ABB RobotStudio station: Vision_HG_20250724-224039.rsstn

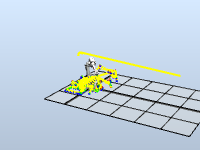
Station Station (saved by RobotStudio 6.8.8148.134)
Controller Vision
  mechanical unit ROB_1: IRB2600_20_165_C_01_2, 6 joints, base frame (0, 0, 0) mm
Layout (positions relative to the parent item):
  - IRB2600_20_165_C_01_2 [mechanism, from Robots\IRB2600_20_165_C_01.rslib] at (0, 0, 0) mm; joint values [-0.7369, -0.204, 0.6129, 0.0001, 1.0987, -0.0243] (rad or m)
  - 框架_2 [frame] at (695.76, -308.93, 242.8) mm, rotated rx -4.43 ry -84.98 rz 46.15 deg
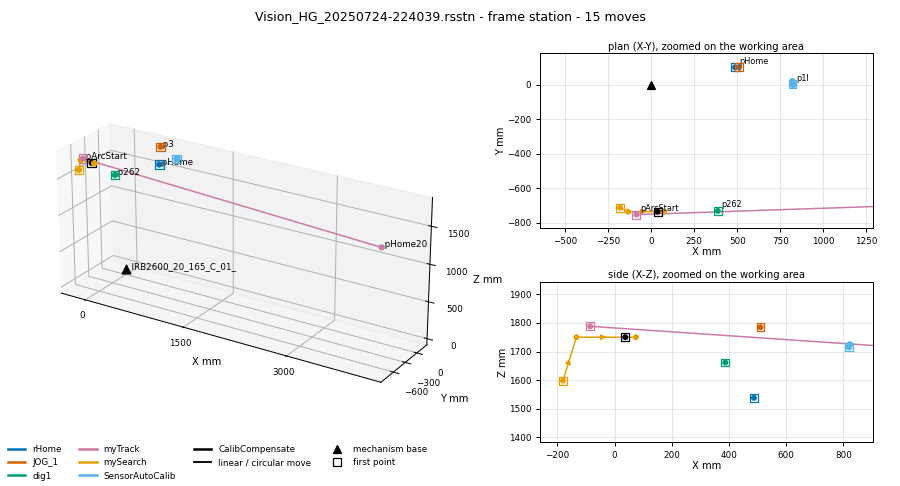
[picture p0: tool path of Vision_HG_20250724-224039.rsstn in frame station, 15 of 295 moves have a stored position in this frame; points joined in program order, loops and branches not executed]
Targets, tools, work objects and paths stored in the station, written as RAPID:
! task T_ROB1
MODULE MainModule
  VAR tooldata p1:=[TRUE,[[0,0,0],[1,0,0,0]],[-1,[0,0,0],[1,0,0,0],0,0,0]];
  LOCAL PERS tooldata p0:=[TRUE,[[0,0,0],[1,0,0,0]],[-1,[0,0,0],[1,0,0,0],0,0,0]];
  PERS tooldata tool3:=[TRUE,[[-77.6624,-1.03018,498.161],[0.800252,-0.0129489,0.0443032,-0.597884]],[10,[79.1,25.2,-267.1],[1,0,0,0],0.143,0.365,0.104]];
  TASK PERS tooldata tool4:=[TRUE,[[0,0,0],[1,0,0,0]],[10,[0,0,0],[1,0,0,0],0,0,0]];
  PERS tooldata tWeldGun:=[TRUE,[[-80.9134,-12.7311,494.27],[0.800252,-0.0129489,0.0443032,-0.597884]],[10,[79.1,25.2,-267.1],[1,0,0,0],0.143,0.365,0.104]];
  PERS tooldata autoCalibRes:=[TRUE,[[-92.3529,67.6081,476.661],[0.14635,-0.09099,-0.47804,-0.86127]],[2,[1,0,0],[1,0,0,0],0,0,0]];
  TASK PERS tooldata tool1:=[TRUE,[[0,0,0],[1,0,0,0]],[-1,[0,0,0],[1,0,0,0],0,0,0]];
  PERS wobjdata wobjcalib:=[FALSE,TRUE,"",[[826.111,71.2533,1714.68],[0.0119558,0.680715,0.732448,-0.00181828]],[[0,0,0],[1,0,0,0]]];
  CONST robtarget pHome:=[[487.33,102.53,1537.96],[0.139151,0.929573,0.0802124,-0.331809],[0,-1,0,1],[165.238,9E+09,9E+09,9E+09,9E+09,9E+09]];
  CONST speeddata speed1:=[25,25,25,25];
  CONST robtarget p3:=[[510.37,102.54,1784.95],[0.139155,0.929576,0.0802308,-0.331793],[0,-1,0,1],[165.238,9E+09,9E+09,9E+09,9E+09,9E+09]];
  CONST robtarget p262:=[[387.21,-731.34,1661.4],[0.0489836,0.0684608,0.2747,-0.957838],[0,0,-1,1],[276.422,9E+09,9E+09,9E+09,9E+09,9E+09]];
  PERS robtarget pArcStart:=[[-85.4083,-752.512,1788.13],[0.0516116,0.0583127,0.355092,-0.931582],[-1,-1,0,1],[443.838,9E+09,9E+09,9E+09,9E+09,9E+09]];
  CONST robtarget pHome20:=[[4100.11,-610.56,1504.11],[0.0519254,0.0584219,0.355084,-0.931561],[-1,-1,-1,1],[4151.67,9E+09,9E+09,9E+09,9E+09,9E+09]];
  CONST robtarget pBegin:=[[-180.6,-712.13,1598.38],[0.0515906,0.0582196,0.355192,-0.931551],[-1,-1,0,1],[443.838,9E+09,9E+09,9E+09,9E+09,9E+09]];
  PERS robtarget pSearchStart:=[[-133.62,-735.71,1750.06],[0.0516116,0.0583127,0.355092,-0.931582],[-1,-1,0,1],[443.838,9E+09,9E+09,9E+09,9E+09,9E+09]];
  PERS robtarget pSearchEnd:=[[74.4,-735.66,1750.11],[0.0517009,0.0583963,0.355037,-0.931593],[-1,-1,0,1],[443.838,9E+09,9E+09,9E+09,9E+09,9E+09]];
  CONST robtarget p1l:=[[-66.95,-10.33,0.38],[0.0609234,-0.0589398,-0.990074,0.112108],[-2,-1,2,1],[1474.6,9E+09,9E+09,9E+09,9E+09,9E+09]];
  CONST robtarget p2l:=[[-56.82,-10.34,0.37],[0.0609473,-0.0589005,-0.990073,0.112123],[-2,-1,2,1],[1474.6,9E+09,9E+09,9E+09,9E+09,9E+09]];
  CONST robtarget p3l:=[[-46.82,-10.3,0.33],[0.0609635,-0.0588963,-0.990075,0.112097],[-2,-1,2,1],[1474.6,9E+09,9E+09,9E+09,9E+09,9E+09]];
  CONST robtarget p1h:=[[-74.01,-7.93,-8.85],[0.0610072,-0.0589652,-0.990068,0.112102],[-2,-1,2,1],[1474.6,9E+09,9E+09,9E+09,9E+09,9E+09]];
  CONST robtarget p2h:=[[-63.94,-7.93,-8.86],[0.0610143,-0.0589296,-0.99007,0.112101],[-2,-1,2,1],[1474.6,9E+09,9E+09,9E+09,9E+09,9E+09]];
  CONST robtarget p3h:=[[-53.65,-7.9,-8.89],[0.0609812,-0.058948,-0.990073,0.112081],[-2,-1,2,1],[1474.6,9E+09,9E+09,9E+09,9E+09,9E+09]];
  CONST robtarget pCompLaser:=[[37.33,-735.63,1750.15],[0.0516795,0.0583772,0.355009,-0.931606],[-1,-1,0,1],[443.838,9E+09,9E+09,9E+09,9E+09,9E+09]];
  PROC main()
    myTrack;
  ENDPROC
  PROC A_Time()
    MoveJ il_16,v500,z50,too11OSPR;
    WaitTime 40;
  ENDPROC
  PROC B_Time()
    MoveJ il_17,v500,z50,too11OSPR;
    WaitTime 40;
  ENDPROC
  PROC rHome()
    MoveL pHome,speed1,z50,tool3;
  ENDPROC
  PROC rInitall()
  ENDPROC
  PROC rWelding()
  ENDPROC
  PROC JOG_1()
    MoveL p3,speed1,z50,tool3;
  ENDPROC
  PROC dig1()
    MoveL p262,speed1,z50,tWeldGun;
  ENDPROC
  PROC myTrack()
    mySearch;
    MoveL pArcStart,speed1,z50,tWeldGun;
    MoveL pHome20,speed1,z50,tWeldGun;
  ENDPROC
  PROC mySearch()
    MoveJ pBegin,v50,fine,tWeldGun;
    MoveL pSearchStart,v50,fine,tWeldGun;
    MoveL pSearchEnd,v20,fine,tWeldGun;
  ENDPROC
  PROC SensorAutoCalib()
    MoveL p1l,v50,fine,tWeldGun\WObj:=wobjcalib;
    MoveL p2l,v50,fine,tWeldGun\WObj:=wobjcalib;
    MoveL p3l,v50,fine,tWeldGun\WObj:=wobjcalib;
    MoveL p1h,v50,fine,tWeldGun\WObj:=wobjcalib;
    MoveL p2h,v50,fine,tWeldGun\WObj:=wobjcalib;
    MoveL p3h,v50,fine,tWeldGun\WObj:=wobjcalib;
    WaitTime 3;
  ENDPROC
  PROC CalibCompensate()
    MoveL pCompLaser,v40,fine,tWeldGun;
    WaitTime 3;
  ENDPROC
  PROC Routine1()
  ENDPROC
  PROC rritest()
    WaitTime 0.5;
  ENDPROC
  PROC rriclose()
  ENDPROC
ENDMODULE

! task T_ROB1
MODULE HG_Vision
  VAR wobjdata Model_1:=[FALSE,TRUE,"",[[0,0,0],[1,0,0,0]],[[0,0,0],[1,0,0,0]]];
  VAR wobjdata Model_2:=[FALSE,TRUE,"",[[695.763,-308.932,242.802],[0.688146,0.238317,-0.632091,0.264803]],[[0,0,0],[1,0,0,0]]];
  PERS tooldata too11OSPR:=[TRUE,[[-150,0,388],[1,0,0,0]],[6,[-150,0,0],[1,0,0,0],0,0,0]];
  PROC HE_Calibration_Demo()
    MoveJ il_1,v400,z50,too11OSPR;
    MoveL il_2,v200,fine,too11OSPR;
    MoveL il_3,v200,fine,too11OSPR;
    MoveL il_4,v200,fine,too11OSPR;
    MoveL il_5,v200,fine,too11OSPR;
    MoveL il_6,v200,fine,too11OSPR;
    MoveL il_7,v200,fine,too11OSPR;
    MoveL il_8,v200,fine,too11OSPR;
    MoveL il_9,v200,fine,too11OSPR;
    MoveL il_10,v200,fine,too11OSPR;
    MoveL il_11,v200,fine,too11OSPR;
    MoveL il_12,v200,fine,too11OSPR;
    MoveL il_13,v200,fine,too11OSPR;
    MoveL il_14,v200,fine,too11OSPR;
    MoveL Calib_Result,v20,fine,too11OSPR;
  ENDPROC
  PROC HE_Creation_Model_Demo()
  ENDPROC
ENDMODULE

! task T_ROB1
MODULE NY_Laser
  PROC B_Line()
    MoveJ il_18,v1000,z30,too11OSPR;
    MoveJ il_19,v1500,fine,too11OSPR;
  ENDPROC
  PROC B_902427()
    MoveJ il_20,v1500,z30,too11OSPR;
    MoveJ il_21,v1500,z30,too11OSPR;
    MoveL il_22,v500,z30,too11OSPR;
    MoveJ il_23,v1500,z30,too11OSPR;
    MoveJ il_24,v500,z30,too11OSPR;
    MoveJ il_25,v500,z30,too11OSPR;
  ENDPROC
  PROC B_952329()
    MoveJ il_26,v1500,z30,too11OSPR;
    MoveJ il_27,v1500,z30,too11OSPR;
    MoveJ il_28,v500,z30,too11OSPR;
    MoveL il_29,v200,z30,too11OSPR;
    MoveJ il_30,v500,z30,too11OSPR;
    MoveJ il_31,v1500,z30,too11OSPR;
  ENDPROC
  PROC B_902430()
    MoveJ il_32,v1500,z30,too11OSPR;
    MoveJ il_33,v1500,z30,too11OSPR;
    MoveL il_34,v500,z30,too11OSPR;
    MoveJ il_35,v1500,z30,too11OSPR;
    MoveJ il_36,v500,z30,too11OSPR;
    MoveJ il_37,v500,z30,too11OSPR;
  ENDPROC
  PROC B_902432()
    MoveJ il_38,v1500,z30,too11OSPR;
    MoveJ il_39,v1500,z30,too11OSPR;
    MoveL il_40,v500,z30,too11OSPR;
    MoveJ il_41,v1500,z30,too11OSPR;
    MoveJ il_42,v1500,z30,too11OSPR;
  ENDPROC
  PROC C_MianBan()
    WaitDI DNDI06,1;
    MoveJ il_43,v1500,z50,too11OSPR;
    MoveJ il_44,v1500,z50,too11OSPR;
    MoveJ il_45,v1500,z50,too11OSPR;
    MoveJ il_46,v1500,z50,too11OSPR;
    MoveJ il_47,v1500,z50,too11OSPR;
    MoveJ il_48,v1500,z50,too11OSPR;
    MoveJ il_49,v1500,z50,too11OSPR;
    MoveJ il_50,v1500,z50,too11OSPR;
    MoveJ il_51,v1500,z50,too11OSPR;
    MoveJ il_52,v1500,z50,too11OSPR;
  ENDPROC
  PROC B_Test()
    MoveJ il_53,v500,z50,too11OSPR;
    MoveJ il_54,v500,z50,too11OSPR;
    MoveJ il_55,v500,z50,too11OSPR;
    MoveJ il_56,v100,z50,too11OSPR;
  ENDPROC
  PROC B_952154()
    MoveJ il_57,v1500,z30,too11OSPR;
    MoveJ il_58,v1500,z30,too11OSPR;
    MoveL il_59,v10,z30,too11OSPR;
    MoveL il_60,v1000,z50,too11OSPR;
    MoveJ il_61,v1000,z50,too11OSPR;
    MoveJ il_62,v1000,z50,too11OSPR;
    MoveL il_63,v1000,z50,too11OSPR;
    MoveJ il_64,v1000,z50,too11OSPR;
    MoveL il_65,v1000,z50,too11OSPR;
    MoveJ il_66,v1000,z50,too11OSPR;
    MoveJ il_67,v1500,z30,too11OSPR;
  ENDPROC
  PROC B_952361()
    MoveJ il_68,v1500,z30,too11OSPR;
    MoveJ il_69,v1500,z30,too11OSPR;
    MoveL il_70,v20,z30,too11OSPR;
    MoveL il_71,v200,z30,too11OSPR;
    MoveL il_72,v10,z30,too11OSPR;
    MoveL il_73,v1000,z50,too11OSPR;
    MoveJ il_74,v1000,z50,too11OSPR;
    MoveJ il_75,v1000,z50,too11OSPR;
    MoveL il_76,v1000,z50,too11OSPR;
    MoveJ il_77,v1000,z50,too11OSPR;
    MoveL il_78,v1000,z50,too11OSPR;
    MoveJ il_79,v1000,z50,too11OSPR;
    MoveJ il_80,v1500,z30,too11OSPR;
  ENDPROC
  PROC A_1_ZJ()
    MoveJ il_81,v500,z50,too11OSPR;
    MoveJ il_82,v500,z50,too11OSPR;
    MoveL il_83,v500,z30,too11OSPR;
    MoveJ il_84,v500,z30,too11OSPR;
  ENDPROC
  PROC A_2_ZJ()
    MoveJ il_85,v500,z50,too11OSPR;
    MoveJ il_86,v500,z50,too11OSPR;
    MoveL il_87,v500,z30,too11OSPR;
    MoveJ il_88,v500,z30,too11OSPR;
  ENDPROC
  PROC B_952329_WB()
    MoveJ il_89,v1500,z30,too11OSPR;
    MoveJ il_90,v1500,z30,too11OSPR;
    MoveL il_91,v20,z30,too11OSPR;
    MoveL il_92,v200,z30,too11OSPR;
    MoveL il_93,v10,z30,too11OSPR;
    MoveL il_94,v1000,z50,too11OSPR;
    MoveJ il_95,v1000,z50,too11OSPR;
    MoveJ il_96,v1000,z50,too11OSPR;
    MoveL il_97,v1000,z50,too11OSPR;
    MoveJ il_98,v1000,z50,too11OSPR;
    MoveL il_99,v1000,z50,too11OSPR;
    MoveJ il_100,v1000,z50,too11OSPR;
    MoveJ il_101,v1500,z30,too11OSPR;
  ENDPROC
  PROC B_YJ()
    SetAO AO1_Laser_Power,1.5;
    MoveJ il_102,v1500,z30,too11OSPR;
    MoveJ il_103,v1500,z30,too11OSPR;
    MoveL il_104,v150,z30,too11OSPR;
    LASER_ON;
    SetAO AO1_Laser_Power,5;
    MoveL il_105,v150,fine,too11OSPR;
    MoveL il_106,v40,z30,too11OSPR;
    MoveL il_107,v40,z30,too11OSPR;
    MoveL il_108,v40,z30,too11OSPR;
    MoveL il_109,v40,z5,too11OSPR;
    MoveC il_110,il_111,v20,z5,too11OSPR;
    MoveL il_112,v30,z5,too11OSPR;
    MoveL il_113,v40,z30,too11OSPR;
    MoveL il_114,v40,z30,too11OSPR;
    MoveL il_115,v40,z30,too11OSPR;
    MoveL il_116,v40,z30,too11OSPR;
    MoveL il_117,v40,z5,too11OSPR;
    MoveC il_118,il_119,v20,z5,too11OSPR;
    MoveL il_120,v30,z5,too11OSPR;
    MoveL il_121,v40,z30,too11OSPR;
    MoveL il_122,v40,z30,too11OSPR;
    MoveL il_123,v40,z30,too11OSPR;
    MoveL il_124,v40,z30,too11OSPR;
    MoveL il_125,v40,z30,too11OSPR;
    MoveL il_126,v40,z5,too11OSPR;
    MoveC il_127,il_128,v20,z5,too11OSPR;
    MoveL il_129,v30,z5,too11OSPR;
    MoveL il_130,v40,z30,too11OSPR;
    MoveL il_131,v40,z30,too11OSPR;
    MoveL il_132,v40,z30,too11OSPR;
    MoveL il_133,v40,z5,too11OSPR;
    MoveC il_134,il_135,v20,z5,too11OSPR;
    MoveL il_136,v30,z5,too11OSPR;
    MoveL il_137,v40,z30,too11OSPR;
    MoveL il_138,v40,z30,too11OSPR;
    MoveL il_139,v40,z5,too11OSPR;
    LASER_OFF;
    MoveJ il_140,v150,z20,too11OSPR;
    MoveJ il_141,v1500,z30,too11OSPR;
  ENDPROC
  PROC Creation_1_RJ()
    MoveJ il_142,v500,z50,too11OSPR;
    MoveJ il_143,v500,z50,too11OSPR;
    MoveJ il_144,v500,z50,too11OSPR;
    MoveL il_145,v200,fine,too11OSPR;
    MoveL il_146,v200,fine,too11OSPR;
    MoveL il_147,v500,z30,too11OSPR;
    MoveJ il_148,v500,z30,too11OSPR;
  ENDPROC
  PROC Creation_2_RJ()
    MoveJ il_149,v500,z50,too11OSPR;
    MoveJ il_150,v500,z50,too11OSPR;
    MoveL il_151,v200,fine,too11OSPR;
    MoveJ il_152,v500,z50,too11OSPR;
    MoveL il_153,v200,fine,too11OSPR;
    MoveL il_154,v500,z30,too11OSPR;
    MoveJ il_155,v500,z30,too11OSPR;
  ENDPROC
  PROC A_Test()
    MoveJ il_156,v1500,z50,too11OSPR;
    MoveL il_157,v200,z50,too11OSPR;
    MoveL il_158,v100,z50,too11OSPR;
    MoveJ il_159,v1500,z50,too11OSPR;
  ENDPROC
  PROC A_1_RJ()
    MoveJ il_160,v500,z50,too11OSPR;
    MoveJ il_161,v500,z50,too11OSPR;
    MoveJ il_162,v500,z50,too11OSPR;
    MoveL il_163,v200,fine,too11OSPR;
    MoveL il_164,v200,fine,too11OSPR;
    MoveL il_165,v500,z30,too11OSPR;
    MoveJ il_166,v500,z30,too11OSPR;
  ENDPROC
  PROC A_2_RJ()
    MoveJ il_167,v500,z50,too11OSPR;
    MoveJ il_168,v500,z50,too11OSPR;
    MoveL il_169,v200,fine,too11OSPR;
    MoveJ il_170,v500,z50,too11OSPR;
    MoveJ il_171,v500,z50,too11OSPR;
    MoveL il_172,v500,z30,too11OSPR;
    MoveJ il_173,v500,z30,too11OSPR;
  ENDPROC
  PROC A_Hezi_Xiao()
    MoveJ il_174,v1000,z50,too11OSPR;
    MoveJ il_175,v1000,z50,too11OSPR;
    MoveL il_176,v500,z50,too11OSPR;
    MoveL il_177,v200,z50,too11OSPR;
    MoveL il_178,v500,z50,too11OSPR;
    MoveJ il_179,v500,z50,too11OSPR;
    MoveJ il_180,v1000,z50,too11OSPR;
  ENDPROC
  PROC A_LongTou()
    MoveJ il_181,v1000,z50,too11OSPR;
    WaitDI DNDI05_Dxu,1;
    MoveL il_182,v500,z50,too11OSPR;
    MoveL il_183,v500,z50,too11OSPR;
    MoveJ il_184,v500,z50,too11OSPR;
  ENDPROC
  PROC A_Cir()
    MoveJ il_185,v1000,z50,too11OSPR;
    MoveL il_186,v500,z50,too11OSPR;
    MoveL il_187,v500,z50,too11OSPR;
    MoveJ il_188,v500,z50,too11OSPR;
    MoveJ il_189,v500,z50,too11OSPR;
    MoveJ il_190,v500,z50,too11OSPR;
    MoveJ il_191,v500,z50,too11OSPR;
    MoveJ il_192,v500,z50,too11OSPR;
  ENDPROC
  PROC B_952364()
    MoveJ il_193,v1500,z30,too11OSPR;
    MoveJ il_194,v1500,z30,too11OSPR;
    MoveL il_195,v20,z30,too11OSPR;
    MoveL il_196,v200,z30,too11OSPR;
    MoveL il_197,v20,z30,too11OSPR;
    MoveL il_198,v1000,z50,too11OSPR;
    MoveJ il_199,v1000,z50,too11OSPR;
    MoveJ il_200,v1000,z50,too11OSPR;
    MoveL il_201,v1000,z50,too11OSPR;
    MoveJ il_202,v1000,z50,too11OSPR;
    MoveL il_203,v1000,z50,too11OSPR;
    MoveJ il_204,v1000,z50,too11OSPR;
    MoveJ il_205,v1500,z30,too11OSPR;
  ENDPROC
  PROC B_902182()
    MoveJ il_206,v1500,z30,too11OSPR;
    MoveJ il_207,v1500,z30,too11OSPR;
    MoveL il_208,v500,z30,too11OSPR;
    MoveJ il_209,v1500,z30,too11OSPR;
    MoveJ il_210,v500,z30,too11OSPR;
    MoveJ il_211,v500,z30,too11OSPR;
  ENDPROC
  PROC B_920282()
    MoveJ il_212,v1500,z30,too11OSPR;
    MoveJ il_213,v1500,z30,too11OSPR;
    MoveL il_214,v500,z30,too11OSPR;
    MoveL il_215,v500,z30,too11OSPR;
    MoveL il_216,v500,z30,too11OSPR;
    MoveL il_217,v500,z30,too11OSPR;
    MoveJ il_218,v1500,z30,too11OSPR;
    MoveJ il_219,v1500,z30,too11OSPR;
  ENDPROC
  PROC A_Hezi()
    MoveJ il_220,v1000,z50,too11OSPR;
    MoveJ il_221,v1000,z50,too11OSPR;
    MoveL il_222,v500,z50,too11OSPR;
    MoveL il_223,v500,z50,too11OSPR;
    MoveJ il_224,v500,z50,too11OSPR;
    MoveJ il_225,v1000,z50,too11OSPR;
  ENDPROC
  PROC B_WeiBian_Text()
    MoveJ il_226,v1500,z30,too11OSPR;
    MoveJ il_227,v1500,z30,too11OSPR;
    MoveL il_228,v500,z30,too11OSPR;
    MoveJ il_229,v1500,z30,too11OSPR;
    MoveJ il_230,v500,z30,too11OSPR;
    MoveJ il_231,v500,z30,too11OSPR;
  ENDPROC
  PROC A_Line()
    MoveJ il_232,v1000,z30,too11OSPR;
    MoveJ il_233,v100,fine,too11OSPR;
    LASER_ON;
    MoveL il_234,v50,fine,too11OSPR;
    LASER_OFF;
  ENDPROC
  PROC B_ZJ()
    SetAO AO1_Laser_Power,6.5;
    MoveJ il_235,v1500,z30,too11OSPR;
    MoveJ il_236,v1500,z30,too11OSPR;
    MoveL il_237,v150,fine,too11OSPR;
    LASER_ON;
    MoveL il_238,v40,z30,too11OSPR;
    MoveL il_239,v40,z30,too11OSPR;
    MoveL il_240,v40,z5,too11OSPR;
    MoveL il_241,v20,fine,too11OSPR;
    LASER_OFF;
    MoveL il_242,v20,fine,too11OSPR;
    LASER_ON;
    MoveL il_243,v20,z1,too11OSPR;
    MoveL il_244,v40,z30,too11OSPR;
    MoveL il_245,v40,z30,too11OSPR;
    MoveL il_246,v40,z5,too11OSPR;
    MoveL il_247,v20,fine,too11OSPR;
    LASER_OFF;
    MoveL il_248,v20,fine,too11OSPR;
    LASER_ON;
    MoveL il_249,v20,fine,too11OSPR;
    MoveL il_250,v40,z30,too11OSPR;
    MoveL il_251,v40,z30,too11OSPR;
    MoveL il_252,v40,z30,too11OSPR;
    MoveL il_253,v40,z30,too11OSPR;
    MoveL il_254,v40,z30,too11OSPR;
    MoveL il_255,v20,fine,too11OSPR;
    LASER_OFF;
    MoveL il_256,v20,fine,too11OSPR;
    LASER_ON;
    MoveL il_257,v20,z1,too11OSPR;
    MoveL il_258,v40,z30,too11OSPR;
    MoveL il_259,v40,z30,too11OSPR;
    MoveL il_260,v40,z5,too11OSPR;
    MoveL il_261,v20,fine,too11OSPR;
    LASER_OFF;
    MoveL il_262,v10,fine,too11OSPR;
    LASER_ON;
    MoveL il_263,v20,z1,too11OSPR;
    MoveL il_264,v40,z30,too11OSPR;
    MoveL il_265,v40,z30,too11OSPR;
    MoveL il_266,v40,z5,too11OSPR;
    LASER_OFF;
    MoveJ il_267,v150,z20,too11OSPR;
    MoveJ il_268,v1500,z30,too11OSPR;
  ENDPROC
ENDMODULE

! task T_ROB1
MODULE NY_DATA
  CONST jointtarget PHOME1:=[[0,0,0,0,90,0],[9E+09,9E+09,9E+09,9E+09,9E+09,9E+09]];
  PROC LASER_ON()
    Set DNDO01_Gas;
    WaitTime 0.15;
    Set DNDO00_Laser;
  ENDPROC
  PROC LASER_OFF()
    Reset DNDO00_Laser;
    WaitTime 0.1;
    Reset DNDO01_Gas;
  ENDPROC
  PROC Pulse()
    SetAO AO1_Laser_Power,1;
    Set DNDO01_Gas;
    PulseDO \PLength:=0.1,DNDO00_Laser;
    WaitTime 0.2;
    Reset DNDO01_Gas;
  ENDPROC
  PROC Zero1()
    MoveAbsJ PHOME1,v100,fine,too11OSPR;
  ENDPROC
ENDMODULE

! task T_ROB1
MODULE MY_weld_track_impl
  PERS tooldata calibRes:=[TRUE,[[0,0,0],[1,0,0,0]],[1,[0,0,0.001],[1,0,0,0],0,0,0]];
  PERS wobjdata obj:=[FALSE,TRUE,"",[[0,0,0],[1,0,0,0]],[[0,0,0],[1,0,0,0]]];
  PROC MY_stop_sensor_impl()
    MY_stop_rri;
    MY_release_thread_resource;
  ENDPROC
  PROC MY_stop_scan_impl()
  ENDPROC
  PROC MY_reduce_corr_impl()
  ENDPROC
  PROC MY_update_robpos_impl()
  ENDPROC
  PROC MY_corr_motion_start_impl()
  ENDPROC
  PROC MY_corr_motion_stop_impl()
  ENDPROC
  PROC MY_search_trap_start_impl()
    MY_init_search_found_trap_imp;
    MY_init_search_timeout_trap_imp;
  ENDPROC
  PROC MY_search_trap_stop_impl()
  ENDPROC
  PROC MY_sensor_close_seam_find_impl()
  ENDPROC
  PROC MY_stop_seam_find_impl()
  ENDPROC
  PROC MY_sensor_calib_get_data_impl()
  ENDPROC
  PROC MY_meas_circle_impl()
  ENDPROC
  PROC MY_calc_plane_impl()
  ENDPROC
  PROC MY_calc_circle_impl()
  ENDPROC
  PROC MY_release_thread_resource()
  ENDPROC
  PROC MY_coord_trans_stop_imp()
    MY_corr_motion_stop_impl;
    PDispOff;
  ENDPROC
  PROC MY_weld_stop_seam_find_imp()
    PDispOff;
  ENDPROC
  PROC MY_init_search_found_trap_imp()
  ENDPROC
  PROC MY_init_search_timeout_trap_imp()
  ENDPROC
  PROC MY_start_rri()
  ENDPROC
  PROC MY_stop_rri()
    WaitTime 1.5;
  ENDPROC
ENDMODULE

! task T_ROB1
MODULE MY_weld_track_intf
  PROC WeldStop()
    MY_coord_trans_stop_imp;
  ENDPROC
  PROC SeamFindStop()
    MY_stop_seam_find_impl;
  ENDPROC
  PROC ScanOff()
    MY_stop_scan_impl;
  ENDPROC
  PROC SensorCalibGetData()
    MY_sensor_calib_get_data_impl;
  ENDPROC
  PROC SeamFindSensorClose()
    MY_sensor_close_seam_find_impl;
  ENDPROC
  PROC MeasCircle()
    MY_meas_circle_impl;
  ENDPROC
  PROC SeamFindStopWeld()
    MY_weld_stop_seam_find_imp;
  ENDPROC
  PROC SensorOff()
    MY_stop_sensor_impl;
  ENDPROC
  PROC ReduceCorr()
    MY_reduce_corr_impl;
  ENDPROC
  PROC CalcCircle()
    MY_calc_circle_impl;
  ENDPROC
  PROC CalcPlane()
    MY_calc_plane_impl;
  ENDPROC
ENDMODULE

! task T_ROB1
MODULE HG_Mes
  PROC HG_Mes_Info_Main()
    HG_Mes_Info_Int;
  ENDPROC
  PROC HG_Mes_Info_Int()
  ENDPROC
ENDMODULE

! task T_ROB1
MODULE HG_Vision
  VAR wobjdata Model_1:=[FALSE,TRUE,"",[[0,0,0],[1,0,0,0]],[[0,0,0],[1,0,0,0]]];
  VAR wobjdata Model_2:=[FALSE,TRUE,"",[[695.763,-308.932,242.802],[0.688146,0.238317,-0.632091,0.264803]],[[0,0,0],[1,0,0,0]]];
  PERS tooldata too11OSPR:=[TRUE,[[-150,0,388],[1,0,0,0]],[6,[-150,0,0],[1,0,0,0],0,0,0]];
  PROC HE_Calibration_Demo()
    MoveJ il_1,v400,z50,too11OSPR;
    MoveL il_2,v200,fine,too11OSPR;
    MoveL il_3,v200,fine,too11OSPR;
    MoveL il_4,v200,fine,too11OSPR;
    MoveL il_5,v200,fine,too11OSPR;
    MoveL il_6,v200,fine,too11OSPR;
    MoveL il_7,v200,fine,too11OSPR;
    MoveL il_8,v200,fine,too11OSPR;
    MoveL il_9,v200,fine,too11OSPR;
    MoveL il_10,v200,fine,too11OSPR;
    MoveL il_11,v200,fine,too11OSPR;
    MoveL il_12,v200,fine,too11OSPR;
    MoveL il_13,v200,fine,too11OSPR;
    MoveL il_14,v200,fine,too11OSPR;
    MoveL Calib_Result,v20,fine,too11OSPR;
  ENDPROC
  PROC HE_Creation_Model_Demo()
  ENDPROC
ENDMODULE

! task T_ROB1
MODULE MainModule
  PROC main()
    HG_Mes_Info_Main;
  ENDPROC
ENDMODULE

! task T_ROB1
MODULE HG_Socket
  PROC Mes_Socket_Info_Receive()
  ENDPROC
ENDMODULE

! task T_ROB1
MODULE HG_Mes
  PROC HG_Mes_Info_Int()
  ENDPROC
  PROC HG_Mes_Info_Main()
    HG_Mes_Info_Int;
  ENDPROC
ENDMODULE

! task T_ROB1
MODULE HG_Laser
  PROC Set_LaserData()
  ENDPROC
ENDMODULE

